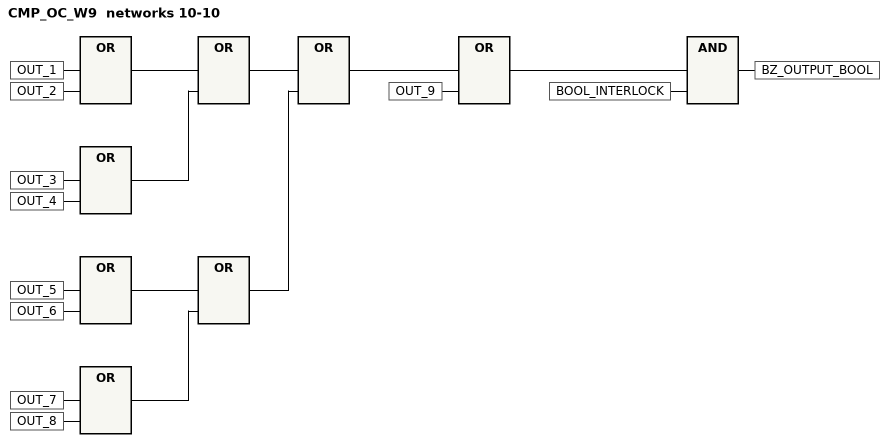
[picture p24: CMP_OC_W9 (FBD) networks 10-10]
_FBD_ (* Function Block Diagram *)
NETWORK 1
	OR(LT(WORD_1, 0), GT(WORD_1, 0)) => OUT_1
NETWORK 2
	OR(LT(WORD_2, 0), GT(WORD_2, 0)) => OUT_2
NETWORK 3
	OR(LT(WORD_3, 0), GT(WORD_3, 0)) => OUT_3
NETWORK 4
	OR(LT(WORD_4, 0), GT(WORD_4, 0)) => OUT_4
NETWORK 5
	OR(LT(WORD_5, 0), GT(WORD_5, 0)) => OUT_5
NETWORK 6
	OR(LT(WORD_6, 0), GT(WORD_6, 0)) => OUT_6
NETWORK 7
	OR(LT(WORD_7, 0), GT(WORD_7, 0)) => OUT_7
NETWORK 8
	OR(LT(WORD_8, 0), GT(WORD_8, 0)) => OUT_8
NETWORK 9
	OR(LT(WORD_9, 0), GT(WORD_9, 0)) => OUT_9
NETWORK 10
	AND(OR(OR(OR(OR(OUT_1, OUT_2), OR(OUT_3, OUT_4)), OR(OR(OUT_5, OUT_6), OR(OUT_7, OUT_8))), OUT_9), BOOL_INTERLOCK) => BZ_OUTPUT_BOOL
_END_FBD_
(* the same logic as Structured Text *)
(* Network 1 *)
OUT_1 := (WORD_1 < 0) OR (WORD_1 > 0);
(* Network 2 *)
OUT_2 := (WORD_2 < 0) OR (WORD_2 > 0);
(* Network 3 *)
OUT_3 := (WORD_3 < 0) OR (WORD_3 > 0);
(* Network 4 *)
OUT_4 := (WORD_4 < 0) OR (WORD_4 > 0);
(* Network 5 *)
OUT_5 := (WORD_5 < 0) OR (WORD_5 > 0);
(* Network 6 *)
OUT_6 := (WORD_6 < 0) OR (WORD_6 > 0);
(* Network 7 *)
OUT_7 := (WORD_7 < 0) OR (WORD_7 > 0);
(* Network 8 *)
OUT_8 := (WORD_8 < 0) OR (WORD_8 > 0);
(* Network 9 *)
OUT_9 := (WORD_9 < 0) OR (WORD_9 > 0);
(* Network 10 *)
BZ_OUTPUT_BOOL := ((((OUT_1 OR OUT_2) OR (OUT_3 OR OUT_4)) OR ((OUT_5 OR OUT_6) OR (OUT_7 OR OUT_8))) OR OUT_9) AND BOOL_INTERLOCK;
END_FUNCTION_BLOCK

(* POU DOWN_COUNT_TIMER, LD *)
FUNCTIONBLOCK DOWN_COUNT_TIMER
VAR_INPUT
	BOOL_SIGNAL_IN: BOOL;
	BOOL_TIMER_RST: BOOL;
	INT_AUTO_RST: INT;
	INT_SV_SEC: INT;
END_VAR
VAR_OUTPUT
	SIGNAL_BOOL: BOOL;
	PV_SEC_INT: INT;
END_VAR
VAR
	DF_1: R_TRIG;
	DF_2: R_TRIG;
	M1: BOOL;
	M2: BOOL;

	T100: TON;
	T101: TON;
	M100: BOOL;
	M101: BOOL;
	M200: BOOL;

	M110: BOOL;
	M300: BOOL;
END_VAR
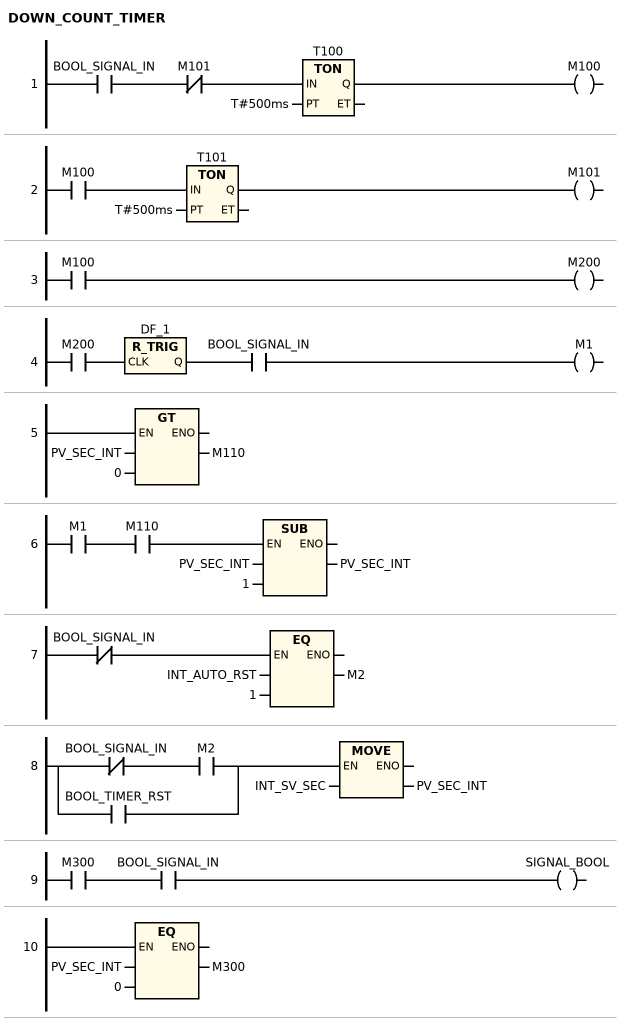
_LD_ (* Ladder Diagram *)
NETWORK 1
	[BOOL_SIGNAL_IN] - [/M101] - T100:TON(IN: *, PT: T#500ms) --- (M100)
NETWORK 2
	[M100] - T101:TON(IN: *, PT: T#500ms) --- (M101)
NETWORK 3
	[M100] --- (M200)
NETWORK 4
	[M200] - DF_1:R_TRIG(CLK: *) - [BOOL_SIGNAL_IN] --- (M1)
NETWORK 5
	*
		EN --- GT(PV_SEC_INT, 0) => M110
NETWORK 6
	[M1] - [M110]
		EN --- SUB(PV_SEC_INT, 1) => PV_SEC_INT
NETWORK 7
	[/BOOL_SIGNAL_IN]
		EN --- EQ(INT_AUTO_RST, 1) => M2
NETWORK 8
	{ [/BOOL_SIGNAL_IN] - [M2] | [BOOL_TIMER_RST] }
		EN --- MOVE(INT_SV_SEC) => PV_SEC_INT
NETWORK 9
	[M300] - [BOOL_SIGNAL_IN] --- (SIGNAL_BOOL)
NETWORK 10
	*
		EN --- EQ(PV_SEC_INT, 0) => M300
_END_LD_
(* the same logic as Structured Text *)
(* Network 1 *)
T100(IN := BOOL_SIGNAL_IN AND NOT M101, PT := T#500ms);
M100 := T100.Q;
(* Network 2 *)
T101(IN := M100, PT := T#500ms);
M101 := T101.Q;
(* Network 3 *)
M200 := M100;
(* Network 4 *)
DF_1(CLK := M200);
M1 := DF_1.Q AND BOOL_SIGNAL_IN;
(* Network 5 *)
M110 := PV_SEC_INT > 0;
(* Network 6 *)
IF M1 AND M110 THEN
	PV_SEC_INT := PV_SEC_INT - 1;
END_IF;
(* Network 7 *)
IF NOT BOOL_SIGNAL_IN THEN
	M2 := INT_AUTO_RST = 1;
END_IF;
(* Network 8 *)
IF NOT BOOL_SIGNAL_IN AND M2 OR BOOL_TIMER_RST THEN
	PV_SEC_INT := INT_SV_SEC;
END_IF;
(* Network 9 *)
SIGNAL_BOOL := M300 AND BOOL_SIGNAL_IN;
(* Network 10 *)
M300 := PV_SEC_INT = 0;
END_FUNCTION_BLOCK

(* POU CLOCK_PLS, LD *)
FUNCTION_BLOCK CLOCK_PLS
VAR_INPUT
	bCpStart			: BOOL;
	INT_TIME_ms 	: INT;

END_VAR
VAR_OUTPUT
	CLOCK_PLS_BOOL: BOOL;
END_VAR
VAR
	T0: TON;
	T1: TON;
	M0: BOOL;
	M1: BOOL;
	D0: TIME;
	D1: TIME;
END_VAR
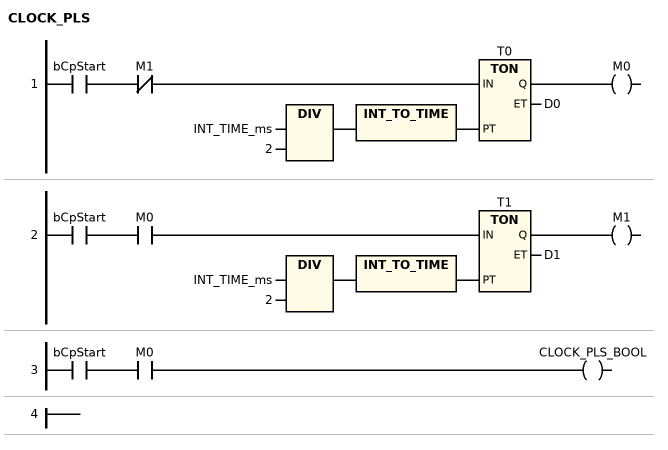
_LD_ (* Ladder Diagram *)
NETWORK 1
	[bCpStart] - [/M1] - T0:TON(IN: *, PT: INT_TO_TIME(DIV(INT_TIME_ms, 2)), ET => D0) --- (M0)
NETWORK 2
	[bCpStart] - [M0] - T1:TON(IN: *, PT: INT_TO_TIME(DIV(INT_TIME_ms, 2)), ET => D1) --- (M1)
NETWORK 3
	[bCpStart] - [M0] --- (CLOCK_PLS_BOOL)
NETWORK 4
	*
_END_LD_
(* the same logic as Structured Text *)
(* Network 1 *)
T0(IN := bCpStart AND NOT M1, PT := INT_TO_TIME(INT_TIME_ms / 2));
D0 := T0.ET;
M0 := T0.Q;
(* Network 2 *)
T1(IN := bCpStart AND M0, PT := INT_TO_TIME(INT_TIME_ms / 2));
D1 := T1.ET;
M1 := T1.Q;
(* Network 3 *)
CLOCK_PLS_BOOL := bCpStart AND M0;
(* Network 4 *)
END_FUNCTION_BLOCK

(* POU DC_PID_FB, LD *)
FUNCTION_BLOCK DC_PID_FB
VAR_INPUT
	BOOL_LOW_FLOW_EN : BOOL;
	INT_HIGH_FLOW_LPM : INT;
	INT_LOW_FLOW_LPM : INT;
	INT_H_L_FLOW_RATIO : INT;
	INT_D1_LPM : INT;
	INT_D2_LPM : INT;
	INT_D3_LPM : INT;
	INT_D4_RAW : INT;
	INT_D5_RAW : INT;
	INT_D6_RAW : INT;
	INT_D1_RATIO : INT;
	INT_D2_RATIO : INT;
	INT_D3_RATIO : INT;
	INT_D4_RATIO : INT;
	INT_D5_RATIO : INT;
	INT_D6_RATIO : INT;

END_VAR

VAR_OUTPUT

	PID_FLOW_RAW : INT;
	D1_RAW_INT : INT;
	D2_RAW_INT : INT;
	D3_RAW_INT : INT;
	D4_LPM_INT : INT;
	D5_LPM_INT : INT;
	D6_LPM_INT : INT;

END_VAR
VAR
	D5EN: BOOL;
	D4EN: BOOL;
	D6EN: BOOL;
	D4REN: BOOL;
	D5REN: BOOL;
	D6REN: BOOL;
END_VAR

(*

Thats 2 program in one function block

1st Program:- 
- Let user able to select High/low flow by trigger bit "BOOL_LOW_FLOW_EN"

	Sequence detail: 
	-If "BOOL_LOW_FLOW_EN" OFF, "INT_HIGH_FLOW_LPM" will MULTIPLY "INT_H_L_FLOW_RATIO" then Feed into "PID_FLOW_RAW".
	-If "BOOL_LOW_FLOW_EN" ON, "INT_LOW_FLOW_LPM" will MULTIPLY "INT_H_L_FLOW_RATIO" then Feed into "PID_FLOW_RAW".
	-"PID_FLOW_RAW should connect direct to ANALOG OUTPUT CARD CHANNEL.


2nd Program:-
-Become Converter. Able to convert 3 types of LPM reading to RAW reading by MULTIPLY the preset RATIO.
-Become Converter. Able to convert 3 types of RAW reading to LPM reading by DIVIDE the preset RATIO.

	Sequence detail:
	-Once detected INT_D1_LPM have value (Not "0") and INT_D1_RATIO have value (Not "0") -> Program will enable and MULTIPLY "INT_D1_LPM" with "INT_D1_RATIO" and feed to "D1_RAW_INT"
	-INT_D2_LPM, INT_D2_RATIO and D2_RAW_INT function same as above (D1)
	-INT_D3_LPM, INT_D3_RATIO and D3_RAW_INT function same as above (D1)
	-Once detected INT_D4_RAW have value (Not "0") and INT_D4_RATIO have value (Not "0") -> Program will enable and DIVIDE "INT_D4_RAW" with "INT_D4_RATIO" and feed to "D4_LPM_INT"
	-INT_D5_RAW, INT_D5_RATIO and D5_LPM_INT function same as above (D4)
	-INT_D6_RAW, INT_D6_RATIO and D6_LPM_INT function same as above (D4)

*)
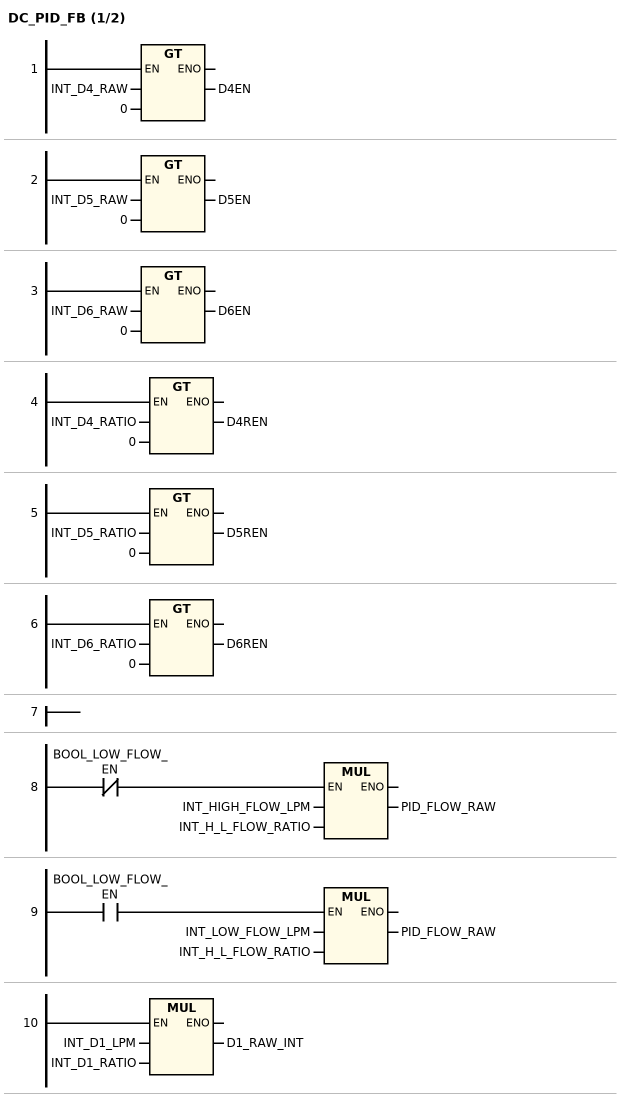
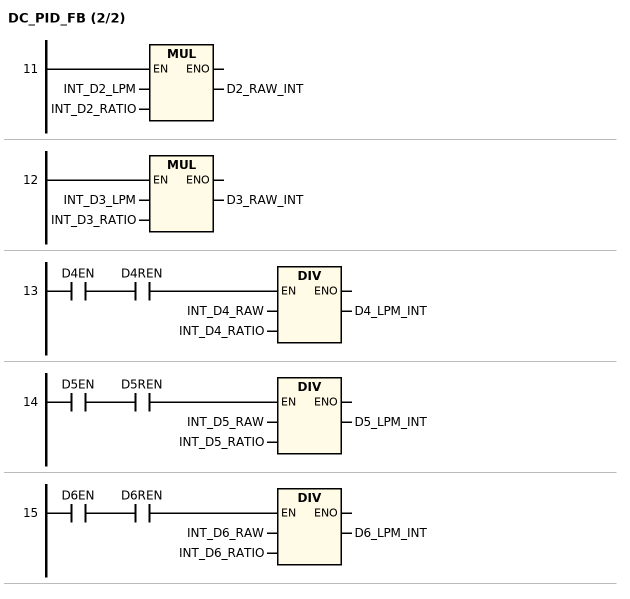
_LD_ (* Ladder Diagram *)
NETWORK 1
	*
		EN --- GT(INT_D4_RAW, 0) => D4EN
NETWORK 2
	*
		EN --- GT(INT_D5_RAW, 0) => D5EN
NETWORK 3
	*
		EN --- GT(INT_D6_RAW, 0) => D6EN
NETWORK 4
	*
		EN --- GT(INT_D4_RATIO, 0) => D4REN
NETWORK 5
	*
		EN --- GT(INT_D5_RATIO, 0) => D5REN
NETWORK 6
	*
		EN --- GT(INT_D6_RATIO, 0) => D6REN
NETWORK 7
	*
NETWORK 8
	[/BOOL_LOW_FLOW_EN]
		EN --- MUL(INT_HIGH_FLOW_LPM, INT_H_L_FLOW_RATIO) => PID_FLOW_RAW
NETWORK 9
	[BOOL_LOW_FLOW_EN]
		EN --- MUL(INT_LOW_FLOW_LPM, INT_H_L_FLOW_RATIO) => PID_FLOW_RAW
NETWORK 10
	*
		EN --- MUL(INT_D1_LPM, INT_D1_RATIO) => D1_RAW_INT
NETWORK 11
	*
		EN --- MUL(INT_D2_LPM, INT_D2_RATIO) => D2_RAW_INT
NETWORK 12
	*
		EN --- MUL(INT_D3_LPM, INT_D3_RATIO) => D3_RAW_INT
NETWORK 13
	[D4EN] - [D4REN]
		EN --- DIV(INT_D4_RAW, INT_D4_RATIO) => D4_LPM_INT
NETWORK 14
	[D5EN] - [D5REN]
		EN --- DIV(INT_D5_RAW, INT_D5_RATIO) => D5_LPM_INT
NETWORK 15
	[D6EN] - [D6REN]
		EN --- DIV(INT_D6_RAW, INT_D6_RATIO) => D6_LPM_INT
_END_LD_
(* the same logic as Structured Text *)
(* Network 1 *)
D4EN := INT_D4_RAW > 0;
(* Network 2 *)
D5EN := INT_D5_RAW > 0;
(* Network 3 *)
D6EN := INT_D6_RAW > 0;
(* Network 4 *)
D4REN := INT_D4_RATIO > 0;
(* Network 5 *)
D5REN := INT_D5_RATIO > 0;
(* Network 6 *)
D6REN := INT_D6_RATIO > 0;
(* Network 7 *)
(* Network 8 *)
IF NOT BOOL_LOW_FLOW_EN THEN
	PID_FLOW_RAW := INT_HIGH_FLOW_LPM * INT_H_L_FLOW_RATIO;
END_IF;
(* Network 9 *)
IF BOOL_LOW_FLOW_EN THEN
	PID_FLOW_RAW := INT_LOW_FLOW_LPM * INT_H_L_FLOW_RATIO;
END_IF;
(* Network 10 *)
D1_RAW_INT := INT_D1_LPM * INT_D1_RATIO;
(* Network 11 *)
D2_RAW_INT := INT_D2_LPM * INT_D2_RATIO;
(* Network 12 *)
D3_RAW_INT := INT_D3_LPM * INT_D3_RATIO;
(* Network 13 *)
IF D4EN AND D4REN THEN
	D4_LPM_INT := INT_D4_RAW / INT_D4_RATIO;
END_IF;
(* Network 14 *)
IF D5EN AND D5REN THEN
	D5_LPM_INT := INT_D5_RAW / INT_D5_RATIO;
END_IF;
(* Network 15 *)
IF D6EN AND D6REN THEN
	D6_LPM_INT := INT_D6_RAW / INT_D6_RATIO;
END_IF;
END_FUNCTION_BLOCK

(* POU EQ_GT, LD *)
FUNCTION_BLOCK EQ_GT
VAR_INPUT
	INT_SOURCE_A: INT;
	INT_SOURCE_B: INT;
END_VAR
VAR_OUTPUT
	SIGNAL_BOOL: BOOL;
END_VAR
VAR
	M0: BOOL;
	M1: BOOL;
END_VAR
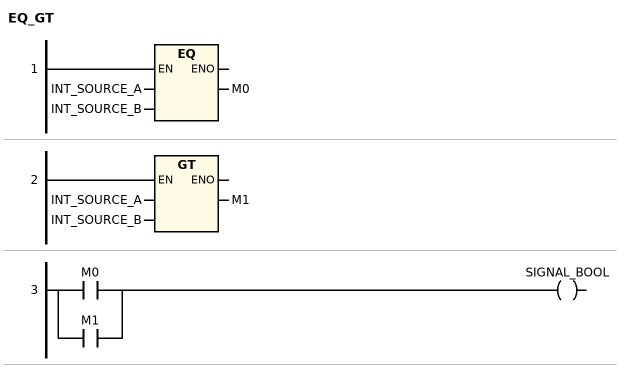
_LD_ (* Ladder Diagram *)
NETWORK 1
	*
		EN --- EQ(INT_SOURCE_A, INT_SOURCE_B) => M0
NETWORK 2
	*
		EN --- GT(INT_SOURCE_A, INT_SOURCE_B) => M1
NETWORK 3
	{ [M0] | [M1] } --- (SIGNAL_BOOL)
_END_LD_
(* the same logic as Structured Text *)
(* Network 1 *)
M0 := INT_SOURCE_A = INT_SOURCE_B;
(* Network 2 *)
M1 := INT_SOURCE_A > INT_SOURCE_B;
(* Network 3 *)
SIGNAL_BOOL := M0 OR M1;
END_FUNCTION_BLOCK

(* POU EQ_LT, LD *)
FUNCTION_BLOCK EQ_LT
VAR_INPUT
	INT_SOURCE_A:INT;
	INT_SOURCE_B:INT;
END_VAR
VAR_OUTPUT
	SIGNAL_BOOL:BOOL;
END_VAR
VAR
	M0: BOOL;
	M1: BOOL;
END_VAR
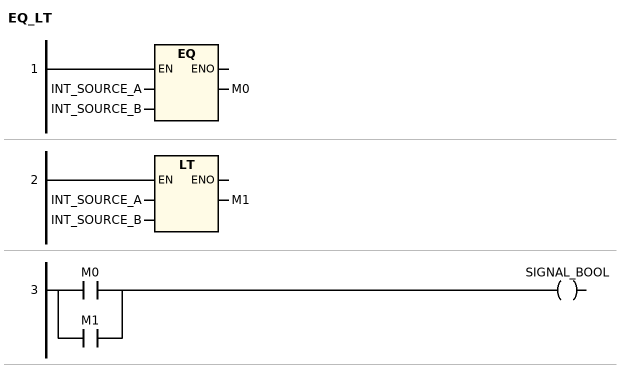
_LD_ (* Ladder Diagram *)
NETWORK 1
	*
		EN --- EQ(INT_SOURCE_A, INT_SOURCE_B) => M0
NETWORK 2
	*
		EN --- LT(INT_SOURCE_A, INT_SOURCE_B) => M1
NETWORK 3
	{ [M0] | [M1] } --- (SIGNAL_BOOL)
_END_LD_
(* the same logic as Structured Text *)
(* Network 1 *)
M0 := INT_SOURCE_A = INT_SOURCE_B;
(* Network 2 *)
M1 := INT_SOURCE_A < INT_SOURCE_B;
(* Network 3 *)
SIGNAL_BOOL := M0 OR M1;
END_FUNCTION_BLOCK

(* POU GUYSON_AI_CTRL, LD *)
FUNCTION_BLOCK GUYSON_AI_CTRL
VAR_INPUT

	BOOL_ST :BOOL; (*Analog Data Collection Start Bit*)
	INT_M1_AI :INT; (*Guyson Generator Master 1 Analog Input Data*)
	INT_M2_AI :INT; (*Guyson Generator Master 2 Analog Input Data*)
	TIME_REFRESH :TIME; (*Refresh Time assigned*)
	TIME_DATA_COLLECT :TIME; (*Delay time for data collection for stability improvement, This data must be ALWAYS "Half" or below from "TIME_REFRESH" SetPoint *)

END_VAR

VAR_OUTPUT

	M1CH1_INT :INT; (*ANALOG READING OF MASTER1-CHANNEL1*)
	M1CH2_INT :INT; (*ANALOG READING OF MASTER1-CHANNEL2*)
	S1CH1_INT :INT; (*ANALOG READING OF SLAVE1-CHANNEL1*)
	M2CH1_INT :INT; (*ANALOG READING OF MASTER2-CHANNEL1*)
	M2CH2_INT :INT; (*ANALOG READING OF MASTER2-CHANNEL2*)
	S2CH1_INT :INT; (*ANALOG READING OF SLAVE2-CHANNEL1*)
	M1_PIN1_DO_BOOL :BOOL; (*GUYSON MASTER 1 SCADA CONNECTOR PIN 1 (A0) CONNECTION OUTPUT FOR MODULE SELECTION*)
	M1_PIN7_DO_BOOL :BOOL; (*GUYSON MASTER 1 SCADA CONNECTOR PIN 7 (A3) CONNECTION OUTPUT FOR IDENTITY SELECTION*)
	M2_PIN1_DO_BOOL :BOOL; (*GUYSON MASTER 2 SCADA CONNECTOR PIN 1 (A0) CONNECTION OUTPUT FOR MODULE SELECTION*)
	M2_PIN7_DO_BOOL :BOOL; (*GUYSON MASTER 2 SCADA CONNECTOR PIN 7 (A3) CONNECTION OUTPUT FOR IDENTITY SELECTION*)
	IT1AOUT_BOOL: BOOL;
	IT2AOUT_BOOL: BOOL;
	IT3AOUT_BOOL: BOOL;
	IT1BOUT_BOOL: BOOL;
	IT2BOUT_BOOL: BOOL;
	IT3BOUT_BOOL: BOOL;





END_VAR
VAR
	IT1A: TON;
	IT2A: TON;
	IT3A: TON;
	IT1B: TON;
	IT2B: TON;
	IT3B: TON;


	M1CH1BOOLOUT: BOOL;
	M1CH2BOOLOUT: BOOL;
	S1CH1BOOLOUT: BOOL;
	M2CH1BOOLOUT: BOOL;
	M2CH2BOOLOUT: BOOL;
	S2CH1BOOLOUT: BOOL;

END_VAR
VAR (* helpers for the ST form of the networks *)
	_p1 : BOOL;
	_p2 : BOOL;
	_p3 : BOOL;
END_VAR
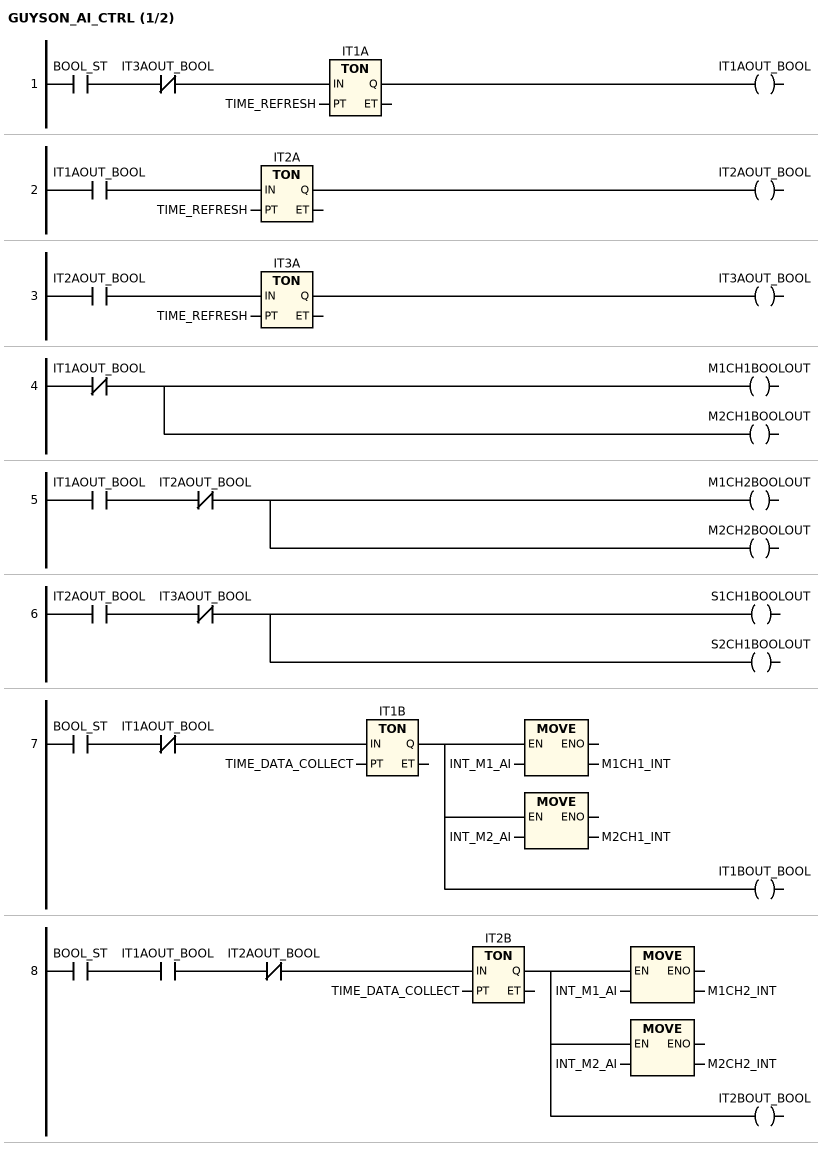
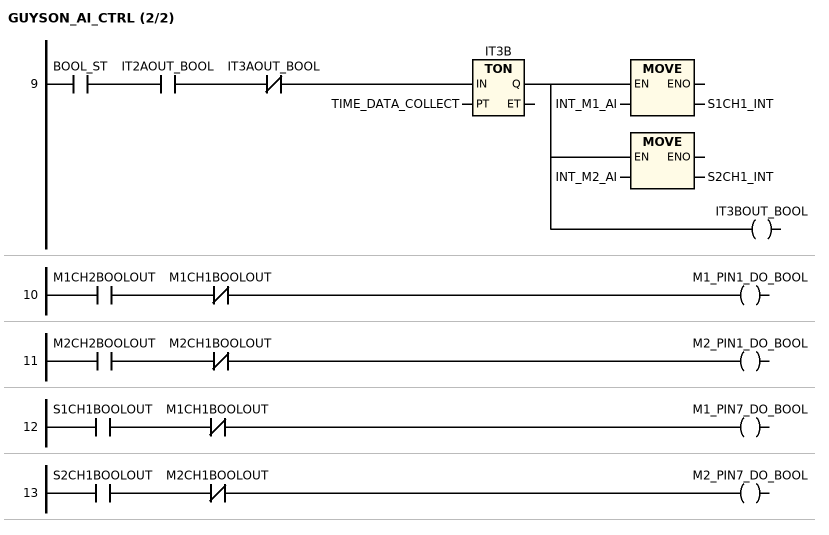
_LD_ (* Ladder Diagram *)
NETWORK 1
	[BOOL_ST] - [/IT3AOUT_BOOL] - IT1A:TON(IN: *, PT: TIME_REFRESH) --- (IT1AOUT_BOOL)
NETWORK 2
	[IT1AOUT_BOOL] - IT2A:TON(IN: *, PT: TIME_REFRESH) --- (IT2AOUT_BOOL)
NETWORK 3
	[IT2AOUT_BOOL] - IT3A:TON(IN: *, PT: TIME_REFRESH) --- (IT3AOUT_BOOL)
NETWORK 4
	[/IT1AOUT_BOOL] --- (M1CH1BOOLOUT) (M2CH1BOOLOUT)
NETWORK 5
	[IT1AOUT_BOOL] - [/IT2AOUT_BOOL] --- (M1CH2BOOLOUT) (M2CH2BOOLOUT)
NETWORK 6
	[IT2AOUT_BOOL] - [/IT3AOUT_BOOL] --- (S1CH1BOOLOUT) (S2CH1BOOLOUT)
NETWORK 7
	[BOOL_ST] - [/IT1AOUT_BOOL] - IT1B:TON(IN: *, PT: TIME_DATA_COLLECT) --- (IT1BOUT_BOOL)
		EN --- MOVE(INT_M1_AI) => M1CH1_INT
		EN --- MOVE(INT_M2_AI) => M2CH1_INT
NETWORK 8
	[BOOL_ST] - [IT1AOUT_BOOL] - [/IT2AOUT_BOOL] - IT2B:TON(IN: *, PT: TIME_DATA_COLLECT) --- (IT2BOUT_BOOL)
		EN --- MOVE(INT_M1_AI) => M1CH2_INT
		EN --- MOVE(INT_M2_AI) => M2CH2_INT
NETWORK 9
	[BOOL_ST] - [IT2AOUT_BOOL] - [/IT3AOUT_BOOL] - IT3B:TON(IN: *, PT: TIME_DATA_COLLECT) --- (IT3BOUT_BOOL)
		EN --- MOVE(INT_M1_AI) => S1CH1_INT
		EN --- MOVE(INT_M2_AI) => S2CH1_INT
NETWORK 10
	[M1CH2BOOLOUT] - [/M1CH1BOOLOUT] --- (M1_PIN1_DO_BOOL)
NETWORK 11
	[M2CH2BOOLOUT] - [/M2CH1BOOLOUT] --- (M2_PIN1_DO_BOOL)
NETWORK 12
	[S1CH1BOOLOUT] - [/M1CH1BOOLOUT] --- (M1_PIN7_DO_BOOL)
NETWORK 13
	[S2CH1BOOLOUT] - [/M2CH1BOOLOUT] --- (M2_PIN7_DO_BOOL)
_END_LD_
(* the same logic as Structured Text *)
(* Network 1 *)
IT1A(IN := BOOL_ST AND NOT IT3AOUT_BOOL, PT := TIME_REFRESH);
IT1AOUT_BOOL := IT1A.Q;
(* Network 2 *)
IT2A(IN := IT1AOUT_BOOL, PT := TIME_REFRESH);
IT2AOUT_BOOL := IT2A.Q;
(* Network 3 *)
IT3A(IN := IT2AOUT_BOOL, PT := TIME_REFRESH);
IT3AOUT_BOOL := IT3A.Q;
(* Network 4 *)
M1CH1BOOLOUT := NOT IT1AOUT_BOOL;
M2CH1BOOLOUT := M1CH1BOOLOUT;
(* Network 5 *)
M1CH2BOOLOUT := IT1AOUT_BOOL AND NOT IT2AOUT_BOOL;
M2CH2BOOLOUT := M1CH2BOOLOUT;
(* Network 6 *)
S1CH1BOOLOUT := IT2AOUT_BOOL AND NOT IT3AOUT_BOOL;
S2CH1BOOLOUT := S1CH1BOOLOUT;
(* Network 7 *)
IT1B(IN := BOOL_ST AND NOT IT1AOUT_BOOL, PT := TIME_DATA_COLLECT);
_p1 := IT1B.Q;
IF _p1 THEN
	M1CH1_INT := INT_M1_AI;
	M2CH1_INT := INT_M2_AI;
END_IF;
IT1BOUT_BOOL := _p1;
(* Network 8 *)
IT2B(IN := BOOL_ST AND IT1AOUT_BOOL AND NOT IT2AOUT_BOOL, PT := TIME_DATA_COLLECT);
_p2 := IT2B.Q;
IF _p2 THEN
	M1CH2_INT := INT_M1_AI;
	M2CH2_INT := INT_M2_AI;
END_IF;
IT2BOUT_BOOL := _p2;
(* Network 9 *)
IT3B(IN := BOOL_ST AND IT2AOUT_BOOL AND NOT IT3AOUT_BOOL, PT := TIME_DATA_COLLECT);
_p3 := IT3B.Q;
IF _p3 THEN
	S1CH1_INT := INT_M1_AI;
	S2CH1_INT := INT_M2_AI;
END_IF;
IT3BOUT_BOOL := _p3;
(* Network 10 *)
M1_PIN1_DO_BOOL := M1CH2BOOLOUT AND NOT M1CH1BOOLOUT;
(* Network 11 *)
M2_PIN1_DO_BOOL := M2CH2BOOLOUT AND NOT M2CH1BOOLOUT;
(* Network 12 *)
M1_PIN7_DO_BOOL := S1CH1BOOLOUT AND NOT M1CH1BOOLOUT;
(* Network 13 *)
M2_PIN7_DO_BOOL := S2CH1BOOLOUT AND NOT M2CH1BOOLOUT;
END_FUNCTION_BLOCK

(* POU GUYSON_AI_RawToWatt, ST *)
FUNCTION_BLOCK GUYSON_AI_RawToWatt
VAR_INPUT

	iAI1raw : INT;				(* 1st Raw Data From Analog Input*)
	iAI2raw : INT;				(* 2nd Raw Data From Analog Input*)
	iAI3raw : INT;				(* 3rd Raw Data From Analog Input*)
	iAI4raw : INT;				(* 4th Raw Data From Analog Input*)
	iAI5raw : INT;				(* 5th Raw Data From Analog Input*)
	iAI6raw : INT;				(* 6th Raw Data From Analog Input*)
	PercentBase : BOOL;		(* The PV will shown Percentage if this Bit is "ON"*)
	WattBase : BOOL;			(* The PV will shown Wattage if this Bit is "ON"*)
	MaxWatt : INT;			(* Defined Max Watt of Generator, Usually is 700W*)

END_VAR
VAR_OUTPUT

	iAI1Value : INT;			(*PV for 1st Data, either Watt or Percent is depend on Base Setting*)
	iAI2Value : INT;			(*PV for 2nd Data, either Watt or Percent is depend on Base Setting*)
	iAI3Value : INT;			(*PV for 3rd Data, either Watt or Percent is depend on Base Setting*)
	iAI4Value : INT;			(*PV for 4th Data, either Watt or Percent is depend on Base Setting*)
	iAI5Value : INT;			(*PV for 5th Data, either Watt or Percent is depend on Base Setting*)
	iAI6Value : INT;			(*PV for 6th Data, either Watt or Percent is depend on Base Setting*)

END_VAR
VAR
	iAI1f: LREAL;
	iAI2f: LREAL;
	iAI3f: LREAL;
	iAI4f: LREAL;
	iAI5f: LREAL;
	iAI6f: LREAL;

	iAI1_Wf: LREAL;
	iAI2_Wf: LREAL;
	iAI3_Wf: LREAL;
	iAI4_Wf: LREAL;
	iAI5_Wf: LREAL;
	iAI6_Wf: LREAL;

	n : INT;

	WRatio: INT;
END_VAR
iAI1f := INT_TO_LREAL (iAI1raw);
iAI2f := INT_TO_LREAL (iAI2raw);
iAI3f := INT_TO_LREAL (iAI3raw);
iAI4f := INT_TO_LREAL (iAI4raw);
iAI5f := INT_TO_LREAL (iAI5raw);
iAI6f := INT_TO_LREAL (iAI6raw);


(*Program to select Watt Base or Percent Base*)

IF PercentBase AND NOT WattBase THEN
n := 11;
END_IF

IF WattBase AND NOT PercentBase THEN
n := 10;
END_IF

IF NOT PercentBase AND NOT WattBase THEN
n := 0;
END_IF

IF PercentBase AND WattBase THEN
n:= 0;
END_IF

CASE n OF

0:; (*No Calculation*)


10: (*Watt Base Calculation *)

iAI1_Wf	:= (iAI1f / 3276.7) * (iAI1f / 3276.7) *20;
iAI2_Wf	:= (iAI2f / 3276.7) * (iAI2f / 3276.7) *20;
iAI3_Wf	:= (iAI3f / 3276.7) * (iAI3f / 3276.7) *20;
iAI4_Wf	:= (iAI4f / 3276.7) * (iAI4f / 3276.7) *20;
iAI5_Wf	:= (iAI5f / 3276.7) * (iAI5f / 3276.7) *20;
iAI6_Wf	:= (iAI6f / 3276.7) * (iAI6f / 3276.7) *20;


11: (*Percent Base Calculation*)


WRatio := MaxWatt/100;


iAI1_Wf	:= ((iAI1f / 3276.7) * (iAI1f / 3276.7) *20)/WRatio;
iAI2_Wf	:= ((iAI2f / 3276.7) * (iAI2f / 3276.7) *20)/WRatio;
iAI3_Wf	:= ((iAI3f / 3276.7) * (iAI3f / 3276.7) *20)/WRatio;
iAI4_Wf	:= ((iAI4f / 3276.7) * (iAI4f / 3276.7) *20)/WRatio;
iAI5_Wf	:= ((iAI5f / 3276.7) * (iAI5f / 3276.7) *20)/WRatio;
iAI6_Wf	:= ((iAI6f / 3276.7) * (iAI6f / 3276.7) *20)/WRatio;

END_CASE

iAI1Value := LREAL_TO_INT (iAI1_Wf);
iAI2Value := LREAL_TO_INT (iAI2_Wf);
iAI3Value := LREAL_TO_INT (iAI3_Wf);
iAI4Value := LREAL_TO_INT (iAI4_Wf);
iAI5Value := LREAL_TO_INT (iAI5_Wf);
iAI6Value := LREAL_TO_INT (iAI6_Wf);
END_FUNCTION_BLOCK

(* POU GUYSON_AI_WattToRaw, ST *)
FUNCTION_BLOCK GUYSON_AI_WattToRaw
VAR_INPUT

	iAI1SP : INT;			(* 1st SetPoint Data*)
	iAI2SP : INT;			(* 2nd SetPoint Data*)
	iAI3SP : INT;			(* 3rd SetPoint Data*)
	iAI4SP : INT;			(* 4th SetPoint Data*)
	iAI5SP : INT;			(* 5th SetPoint Data*)
	iAI6SP : INT;			(* 6th SetPoint Data*)
	PercentBase : BOOL;	(* The PV will shown Percentage if this Bit is "ON"*)
	WattBase: BOOL;		(* The PV will shown Wattage if this Bit is "ON"*)
	MinSP : INT;			(* Define Min SetPoint Input, if SP set below this value, the PV will become "0"*)
	MaxSP : INT;			(* Define Max SetPoint Input, if SP set Greater than value, the PV will become "0"*)
	MaxWatt : INT;		(* Defined Max Watt of Generator, Usually is 700W*)


END_VAR

VAR_OUTPUT

	iAI1raw : INT;			(*1st Raw Data to feed to Analog Output Card for Ultrasonic Generator Power Control*)
	iAI2raw : INT;			(*2nd Raw Data to feed to Analog Output Card for Ultrasonic Generator Power Control*)
	iAI3raw : INT;			(*3rd Raw Data to feed to Analog Output Card for Ultrasonic Generator Power Control*)
	iAI4raw : INT;			(*4th Raw Data to feed to Analog Output Card for Ultrasonic Generator Power Control*)
	iAI5raw : INT;			(*5th Raw Data to feed to Analog Output Card for Ultrasonic Generator Power Control*)
	iAI6raw : INT;			(*6th Raw Data to feed to Analog Output Card for Ultrasonic Generator Power Control*)

END_VAR
VAR
	iAI1f: LREAL;
	iAI2f: LREAL;
	iAI3f: LREAL;
	iAI4f: LREAL;
	iAI5f: LREAL;
	iAI6f: LREAL;

	iAI1_Wf: LREAL;
	iAI2_Wf: LREAL;
	iAI3_Wf: LREAL;
	iAI4_Wf: LREAL;
	iAI5_Wf: LREAL;
	iAI6_Wf: LREAL;

	n : INT;
	WRatio: INT;
END_VAR
(*Set Min and Max Limit for Watt input*)
(*Convert INT to LREAL for Calculation*)

IF iAI1SP>=MinSP AND iAI1SP<=MaxSP THEN
iAI1_Wf := INT_TO_LREAL (iAI1SP);
ELSE iAI1_Wf := 0;
END_IF

IF iAI2SP>=MinSP AND iAI2SP<=MaxSP THEN
iAI2_Wf := INT_TO_LREAL (iAI2SP);
ELSE iAI2_Wf := 0;
END_IF

IF iAI3SP>=MinSP AND iAI3SP<=MaxSP THEN
iAI3_Wf := INT_TO_LREAL (iAI3SP);
ELSE iAI3_Wf := 0;
END_IF

IF iAI4SP>=MinSP AND iAI4SP<=MaxSP THEN
iAI4_Wf := INT_TO_LREAL (iAI4SP);
ELSE iAI4_Wf := 0;
END_IF

IF iAI5SP>=MinSP AND iAI5SP<=MaxSP THEN
iAI5_Wf := INT_TO_LREAL (iAI5SP);
ELSE iAI5_Wf := 0;
END_IF

IF iAI6SP>=MinSP AND iAI6SP<=MaxSP THEN
iAI6_Wf := INT_TO_LREAL (iAI6SP);
ELSE iAI6_Wf := 0;
END_IF

(*Program to select Watt Base or Percent Base*)

IF PercentBase AND NOT WattBase THEN
n := 11;
END_IF

IF WattBase AND NOT PercentBase THEN
n := 10;
END_IF

IF NOT PercentBase AND NOT WattBase THEN
n := 0;
END_IF

IF PercentBase AND WattBase THEN
n:= 0;
END_IF



CASE n OF

0:;	(*No Calculation Apply*)

10:	(*Watt Base Calculation*)

WRatio := MaxWatt/100;


	iAI1f	:= iAI1_Wf/WRatio*327.67;
	iAI2f	:= iAI2_Wf/WRatio*327.67;
	iAI3f	:= iAI3_Wf/WRatio*327.67;
	iAI4f	:= iAI4_Wf/WRatio*327.67;
	iAI5f	:= iAI5_Wf/WRatio*327.67;
	iAI6f	:= iAI6_Wf/WRatio*327.67;


(*	iAI1f	:= (SQRT(iAI1_Wf/20))*3276.7;
	iAI2f	:= (SQRT(iAI2_Wf/20))*3276.7;
	iAI3f	:= (SQRT(iAI3_Wf/20))*3276.7;
	iAI4f	:= (SQRT(iAI4_Wf/20))*3276.7;
	iAI5f	:= (SQRT(iAI5_Wf/20))*3276.7;
	iAI6f	:= (SQRT(iAI6_Wf/20))*3276.7;
*)

11: 	(*% Base Calculation*)

	iAI1f	:= iAI1_Wf*327.67;
	iAI2f	:= iAI2_Wf*327.67;
	iAI3f	:= iAI3_Wf*327.67;
	iAI4f	:= iAI4_Wf*327.67;
	iAI5f	:= iAI5_Wf*327.67;
	iAI6f	:= iAI6_Wf*327.67;

END_CASE

iAI1raw := LREAL_TO_INT (iAI1f);
iAI2raw := LREAL_TO_INT (iAI2f);
iAI3raw := LREAL_TO_INT (iAI3f);
iAI4raw := LREAL_TO_INT (iAI4f);
iAI5raw := LREAL_TO_INT (iAI5f);
iAI6raw := LREAL_TO_INT (iAI6f);
END_FUNCTION_BLOCK

(* POU GUYSON_PRG_SEL, FBD *)
FUNCTION_BLOCK GUYSON_PRG_SEL
VAR_INPUT

	US_ON_BOOL		:BOOL; 		(*ULTRASONIC ON/OFF BIT*)
	PRG_ADD_INT		:INT;		(*PROGRAM ADDRESS*)


END_VAR
VAR_OUTPUT

	BOOL_US_BIT1		:BOOL; 		(*ULTRASONIC EXT1*)
	BOOL_US_BIT2		:BOOL; 		(*ULTRASONIC EXT2*)
	BOOL_US_BIT3		:BOOL; 		(*ULTRASONIC EXT3*)


END_VAR
VAR
END_VAR
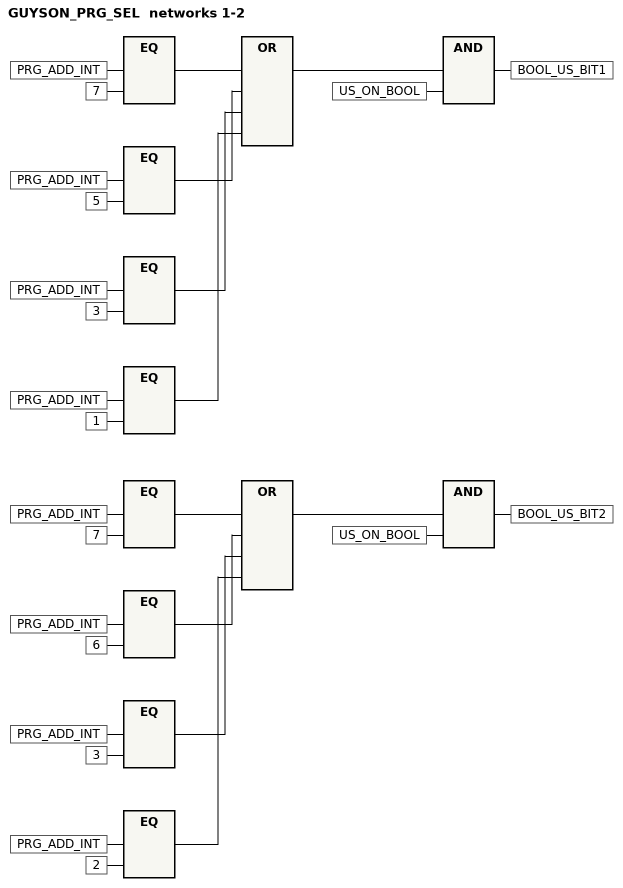
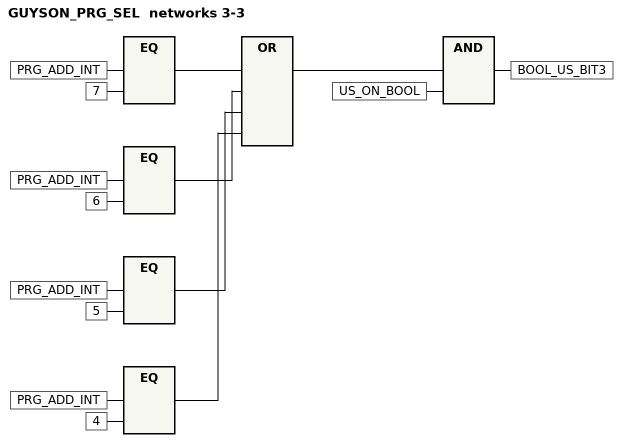
_FBD_ (* Function Block Diagram *)
NETWORK 1
	AND(OR(EQ(PRG_ADD_INT, 7), EQ(PRG_ADD_INT, 5), EQ(PRG_ADD_INT, 3), EQ(PRG_ADD_INT, 1)), US_ON_BOOL) => BOOL_US_BIT1
NETWORK 2
	AND(OR(EQ(PRG_ADD_INT, 7), EQ(PRG_ADD_INT, 6), EQ(PRG_ADD_INT, 3), EQ(PRG_ADD_INT, 2)), US_ON_BOOL) => BOOL_US_BIT2
NETWORK 3
	AND(OR(EQ(PRG_ADD_INT, 7), EQ(PRG_ADD_INT, 6), EQ(PRG_ADD_INT, 5), EQ(PRG_ADD_INT, 4)), US_ON_BOOL) => BOOL_US_BIT3
_END_FBD_
(* the same logic as Structured Text *)
(* Network 1 *)
BOOL_US_BIT1 := ((PRG_ADD_INT = 7) OR (PRG_ADD_INT = 5) OR (PRG_ADD_INT = 3) OR (PRG_ADD_INT = 1)) AND US_ON_BOOL;
(* Network 2 *)
BOOL_US_BIT2 := ((PRG_ADD_INT = 7) OR (PRG_ADD_INT = 6) OR (PRG_ADD_INT = 3) OR (PRG_ADD_INT = 2)) AND US_ON_BOOL;
(* Network 3 *)
BOOL_US_BIT3 := ((PRG_ADD_INT = 7) OR (PRG_ADD_INT = 6) OR (PRG_ADD_INT = 5) OR (PRG_ADD_INT = 4)) AND US_ON_BOOL;
END_FUNCTION_BLOCK

(* POU INDIRECT_FN, LD *)
FUNCTION_BLOCK INDIRECT_FN
VAR_INPUT
	BOOL_SV_PB: BOOL;		(*SAVE PB (TS)*)
	BOOL_LD_PB: BOOL;			(*LOAD PB (TS)*)
	INT_P_NO: INT;		(*PROGRAM NO (TS) 1~10*)
	INT_D00:INT;
	INT_D01:INT;
	INT_D02:INT;
	INT_D03:INT;
	INT_D04:INT;
	INT_D05:INT;
	INT_D06:INT;
	INT_D07:INT;
	INT_D08:INT;
	INT_D09:INT;
	INT_D10:INT;
	INT_D11:INT;
	INT_D12:INT;
	INT_D13:INT;
	INT_D14:INT;
	INT_D15:INT;
	INT_D16:INT;
	INT_D17:INT;
	INT_D18:INT;
	INT_D19:INT;
	INT_D20:INT;
	INT_D21:INT;
	INT_D22:INT;
	INT_D23:INT;
	INT_D24:INT;
	INT_D25:INT;
	INT_D26:INT;
	INT_D27:INT;
	INT_D28:INT;
	INT_D29:INT;
	INT_D30:INT;
	STG_STG1:STRING;
END_VAR
VAR_OUTPUT
	SV_PB_IND_BOOL:BOOL;
	LD_PB_IND_BOOL:BOOL;
	D00_INT:INT;
	D01_INT:INT;
	D02_INT:INT;
	D03_INT:INT;
	D04_INT:INT;
	D05_INT:INT;
	D06_INT:INT;
	D07_INT:INT;
	D08_INT:INT;
	D09_INT:INT;
	D10_INT:INT;
	D11_INT:INT;
	D12_INT:INT;
	D13_INT:INT;
	D14_INT:INT;
	D15_INT:INT;
	D16_INT:INT;
	D17_INT:INT;
	D18_INT:INT;
	D19_INT:INT;
	D20_INT:INT;
	D21_INT:INT;
	D22_INT:INT;
	D23_INT:INT;
	D24_INT:INT;
	D25_INT:INT;
	D26_INT:INT;
	D27_INT:INT;
	D28_INT:INT;
	D29_INT:INT;
	D30_INT:INT;
	STG1_STG:STRING;
END_VAR
VAR

	P1B: BOOL;
	P2B: BOOL;
	P3B: BOOL;
	P4B: BOOL;
	P5B: BOOL;
	P6B: BOOL;
	P7B: BOOL;
	P8B: BOOL;
	P9B: BOOL;
	P10B: BOOL;
	SV_HR: BOOL;
	SV_T: TON;
	SV_CR: BOOL;
	LD_HR: BOOL;
	LD_CR: BOOL;
	LD_T: TON;
	SV_DF: R_TRIG;
	SV_PLS: BOOL;
	LD_DF: R_TRIG;
	LD_PLS: BOOL;
	ALWAYS_ON: BOOL;
	TPC: TON;
	N0: BOOL;
	TPC1: TON;
	N1: BOOL;
	CNG_P_NO: INT;
	NPC: BOOL;		(*NON PROGRAM CHANGE*)
	PCDF: R_TRIG;
	PCTDF: BOOL;
	PCDFN: F_TRIG;
	PC_PLS: BOOL;
	SVPLS: R_TRIG;
	SV_PB_PLS: BOOL;
	LDPLS: R_TRIG;
	LD_PB_PLS: BOOL;
END_VAR
VAR PERSISTENT
	P01D00:INT;
	P01D01:INT;
	P01D02:INT;
	P01D03:INT;
	P01D04:INT;
	P01D05:INT;
	P01D06:INT;
	P01D07:INT;
	P01D08:INT;
	P01D09:INT;
	P01D10:INT;
	P01D11:INT;
	P01D12:INT;
	P01D13:INT;
	P01D14:INT;
	P01D15:INT;
	P01D16:INT;
	P01D17:INT;
	P01D18:INT;
	P01D19:INT;
	P01D20:INT;
	P01D21:INT;
	P01D22:INT;
	P01D23:INT;
	P01D24:INT;
	P01D25:INT;
	P01D26:INT;
	P01D27:INT;
	P01D28:INT;
	P01D29:INT;
	P01D30:INT;
	P01STG:STRING;
	P02D00:INT;
	P02D01:INT;
	P02D02:INT;
	P02D03:INT;
	P02D04:INT;
	P02D05:INT;
	P02D06:INT;
	P02D07:INT;
	P02D08:INT;
	P02D09:INT;
	P02D10:INT;
	P02D11:INT;
	P02D12:INT;
	P02D13:INT;
	P02D14:INT;
	P02D15:INT;
	P02D16:INT;
	P02D17:INT;
	P02D18:INT;
	P02D19:INT;
	P02D20:INT;
	P02D21:INT;
	P02D22:INT;
	P02D23:INT;
	P02D24:INT;
	P02D25:INT;
	P02D26:INT;
	P02D27:INT;
	P02D28:INT;
	P02D29:INT;
	P02D30:INT;
	P02STG:STRING;
	P03D00:INT;
	P03D01:INT;
	P03D02:INT;
	P03D03:INT;
	P03D04:INT;
	P03D05:INT;
	P03D06:INT;
	P03D07:INT;
	P03D08:INT;
	P03D09:INT;
	P03D10:INT;
	P03D11:INT;
	P03D12:INT;
	P03D13:INT;
	P03D14:INT;
	P03D15:INT;
	P03D16:INT;
	P03D17:INT;
	P03D18:INT;
	P03D19:INT;
	P03D20:INT;
	P03D21:INT;
	P03D22:INT;
	P03D23:INT;
	P03D24:INT;
	P03D25:INT;
	P03D26:INT;
	P03D27:INT;
	P03D28:INT;
	P03D29:INT;
	P03D30:INT;
	P03STG:STRING;
	P04D00:INT;
	P04D01:INT;
	P04D02:INT;
	P04D03:INT;
	P04D04:INT;
	P04D05:INT;
	P04D06:INT;
	P04D07:INT;
	P04D08:INT;
	P04D09:INT;
	P04D10:INT;
	P04D11:INT;
	P04D12:INT;
	P04D13:INT;
	P04D14:INT;
	P04D15:INT;
	P04D16:INT;
	P04D17:INT;
	P04D18:INT;
	P04D19:INT;
	P04D20:INT;
	P04D21:INT;
	P04D22:INT;
	P04D23:INT;
	P04D24:INT;
	P04D25:INT;
	P04D26:INT;
	P04D27:INT;
	P04D28:INT;
	P04D29:INT;
	P04D30:INT;
	P04STG:STRING;
	P05D00:INT;
	P05D01:INT;
	P05D02:INT;
	P05D03:INT;
	P05D04:INT;
	P05D05:INT;
	P05D06:INT;
	P05D07:INT;
	P05D08:INT;
	P05D09:INT;
	P05D10:INT;
	P05D11:INT;
	P05D12:INT;
	P05D13:INT;
	P05D14:INT;
	P05D15:INT;
	P05D16:INT;
	P05D17:INT;
	P05D18:INT;
	P05D19:INT;
	P05D20:INT;
	P05D21:INT;
	P05D22:INT;
	P05D23:INT;
	P05D24:INT;
	P05D25:INT;
	P05D26:INT;
	P05D27:INT;
	P05D28:INT;
	P05D29:INT;
	P05D30:INT;
	P05STG:STRING;
	P06D00:INT;
	P06D01:INT;
	P06D02:INT;
	P06D03:INT;
	P06D04:INT;
	P06D05:INT;
	P06D06:INT;
	P06D07:INT;
	P06D08:INT;
	P06D09:INT;
	P06D10:INT;
	P06D11:INT;
	P06D12:INT;
	P06D13:INT;
	P06D14:INT;
	P06D15:INT;
	P06D16:INT;
	P06D17:INT;
	P06D18:INT;
	P06D19:INT;
	P06D20:INT;
	P06D21:INT;
	P06D22:INT;
	P06D23:INT;
	P06D24:INT;
	P06D25:INT;
	P06D26:INT;
	P06D27:INT;
	P06D28:INT;
	P06D29:INT;
	P06D30:INT;
	P06STG:STRING;
	P07D00:INT;
	P07D01:INT;
	P07D02:INT;
	P07D03:INT;
	P07D04:INT;
	P07D05:INT;
	P07D06:INT;
	P07D07:INT;
	P07D08:INT;
	P07D09:INT;
	P07D10:INT;
	P07D11:INT;
	P07D12:INT;
	P07D13:INT;
	P07D14:INT;
	P07D15:INT;
	P07D16:INT;
	P07D17:INT;
	P07D18:INT;
	P07D19:INT;
	P07D20:INT;
	P07D21:INT;
	P07D22:INT;
	P07D23:INT;
	P07D24:INT;
	P07D25:INT;
	P07D26:INT;
	P07D27:INT;
	P07D28:INT;
	P07D29:INT;
	P07D30:INT;
	P07STG:STRING;
	P08D00:INT;
	P08D01:INT;
	P08D02:INT;
	P08D03:INT;
	P08D04:INT;
	P08D05:INT;
	P08D06:INT;
	P08D07:INT;
	P08D08:INT;
	P08D09:INT;
	P08D10:INT;
	P08D11:INT;
	P08D12:INT;
	P08D13:INT;
	P08D14:INT;
	P08D15:INT;
	P08D16:INT;
	P08D17:INT;
	P08D18:INT;
	P08D19:INT;
	P08D20:INT;
	P08D21:INT;
	P08D22:INT;
	P08D23:INT;
	P08D24:INT;
	P08D25:INT;
	P08D26:INT;
	P08D27:INT;
	P08D28:INT;
	P08D29:INT;
	P08D30:INT;
	P08STG:STRING;
	P09D00:INT;
	P09D01:INT;
	P09D02:INT;
	P09D03:INT;
	P09D04:INT;
	P09D05:INT;
	P09D06:INT;
	P09D07:INT;
	P09D08:INT;
	P09D09:INT;
	P09D10:INT;
	P09D11:INT;
	P09D12:INT;
	P09D13:INT;
	P09D14:INT;
	P09D15:INT;
	P09D16:INT;
	P09D17:INT;
	P09D18:INT;
	P09D19:INT;
	P09D20:INT;
	P09D21:INT;
	P09D22:INT;
	P09D23:INT;
	P09D24:INT;
	P09D25:INT;
	P09D26:INT;
	P09D27:INT;
	P09D28:INT;
	P09D29:INT;
	P09D30:INT;
	P09STG:STRING;
	P10D00:INT;
	P10D01:INT;
	P10D02:INT;
	P10D03:INT;
	P10D04:INT;
	P10D05:INT;
	P10D06:INT;
	P10D07:INT;
	P10D08:INT;
	P10D09:INT;
	P10D10:INT;
	P10D11:INT;
	P10D12:INT;
	P10D13:INT;
	P10D14:INT;
	P10D15:INT;
	P10D16:INT;
	P10D17:INT;
	P10D18:INT;
	P10D19:INT;
	P10D20:INT;
	P10D21:INT;
	P10D22:INT;
	P10D23:INT;
	P10D24:INT;
	P10D25:INT;
	P10D26:INT;
	P10D27:INT;
	P10D28:INT;
	P10D29:INT;
	P10D30:INT;
	P10STG:STRING;

END_VAR
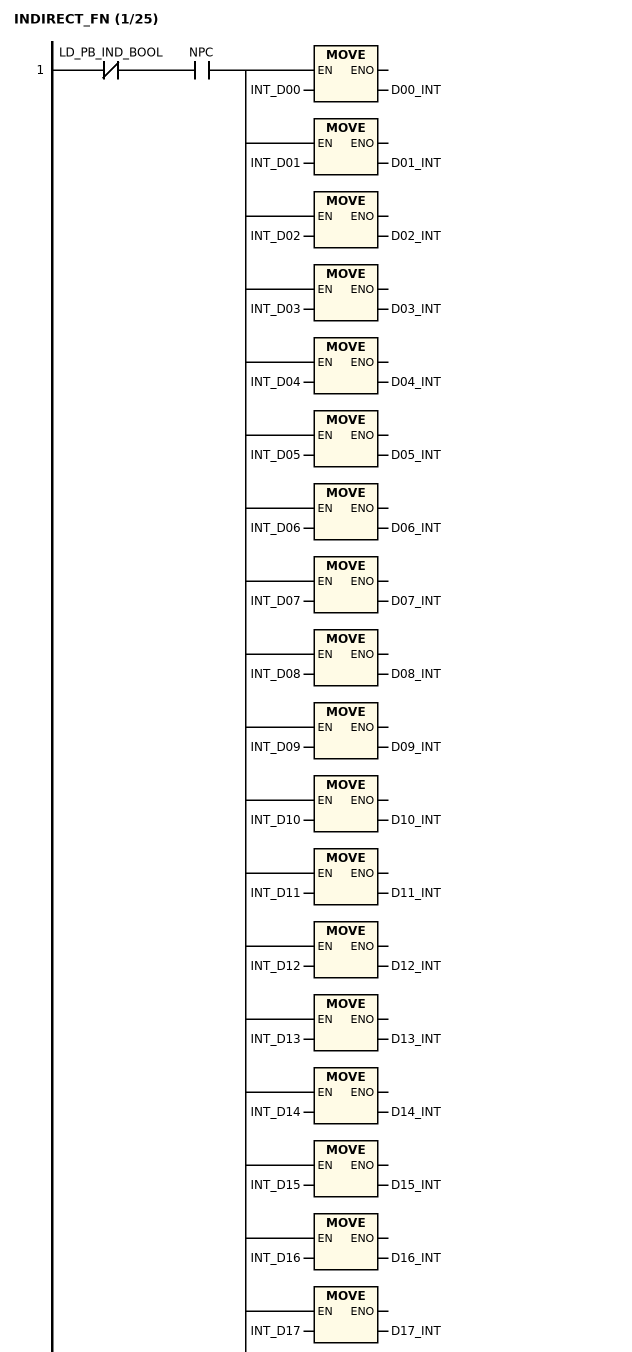
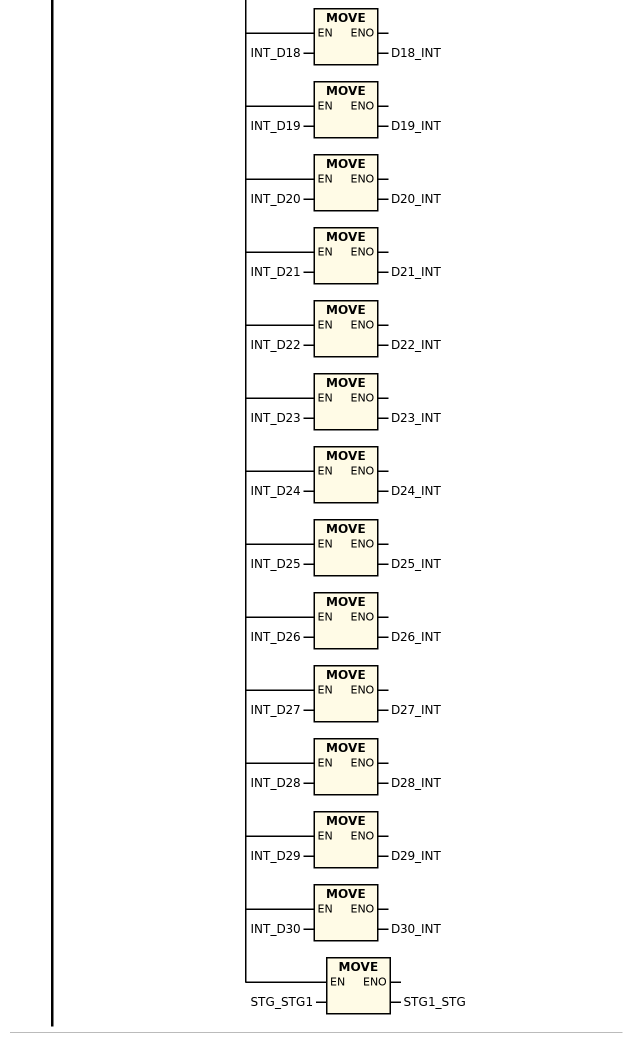
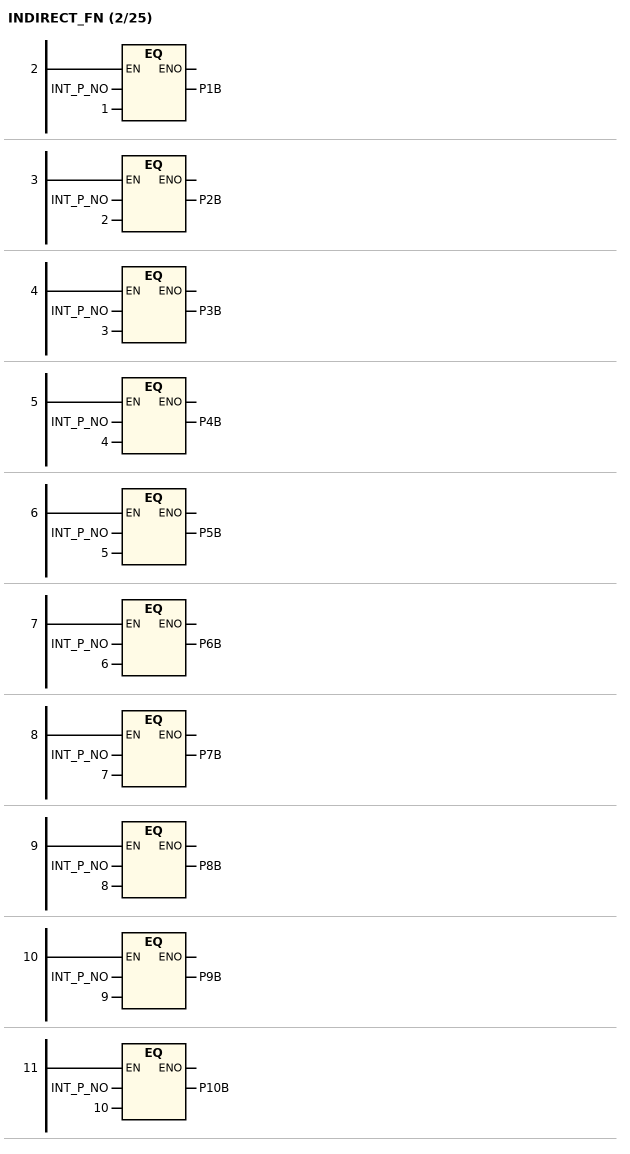
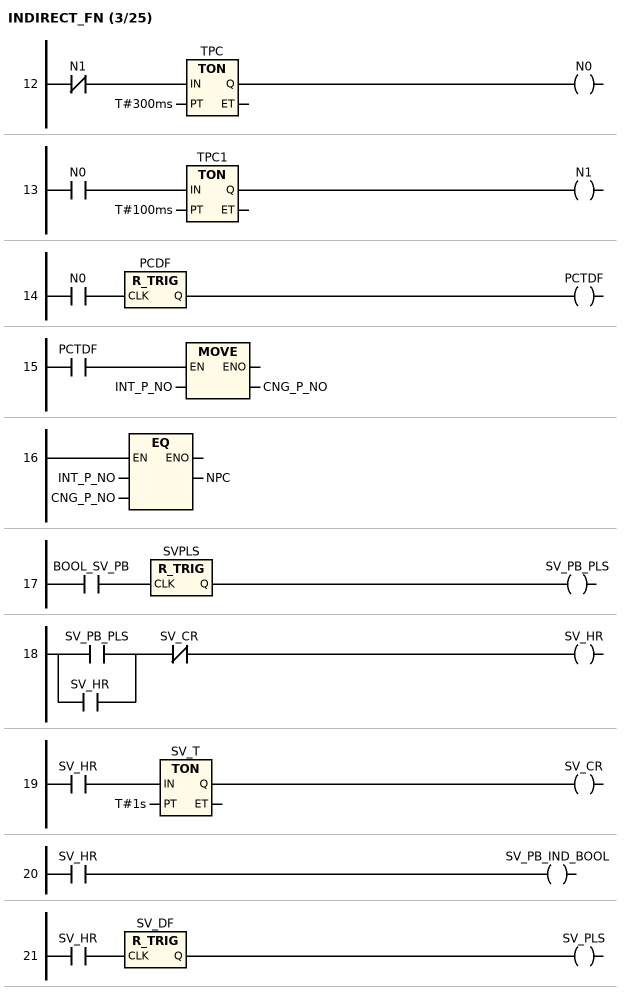
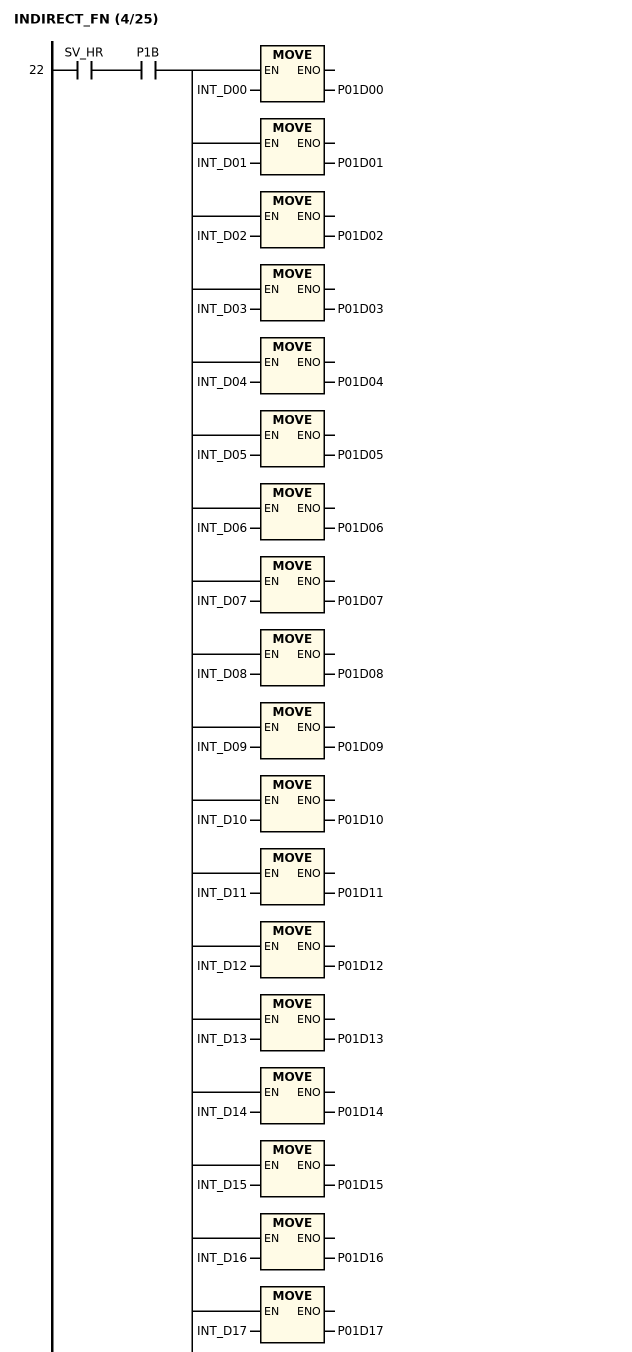
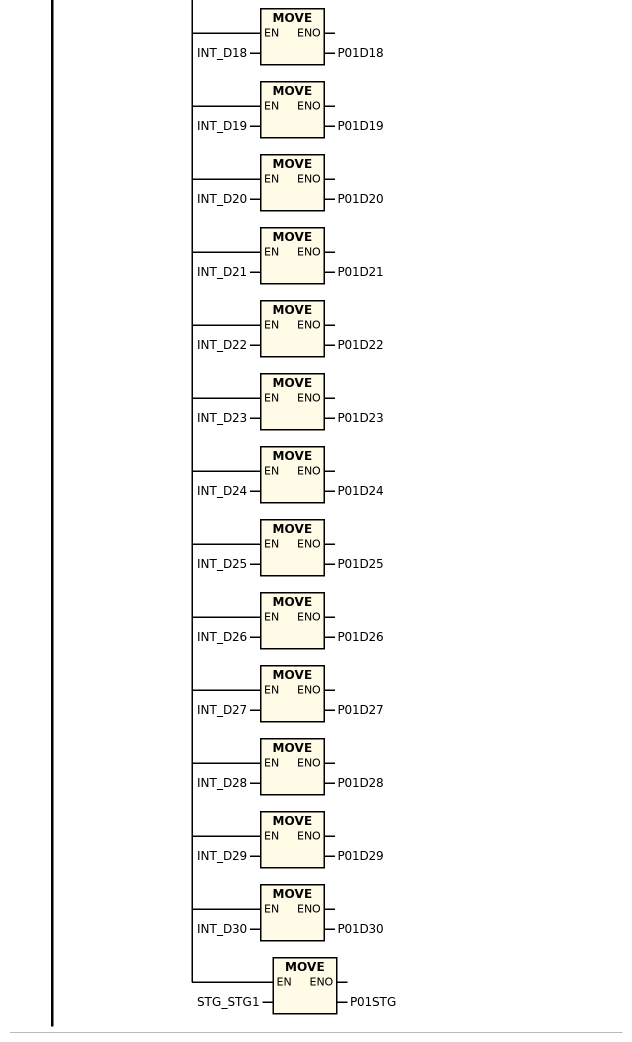
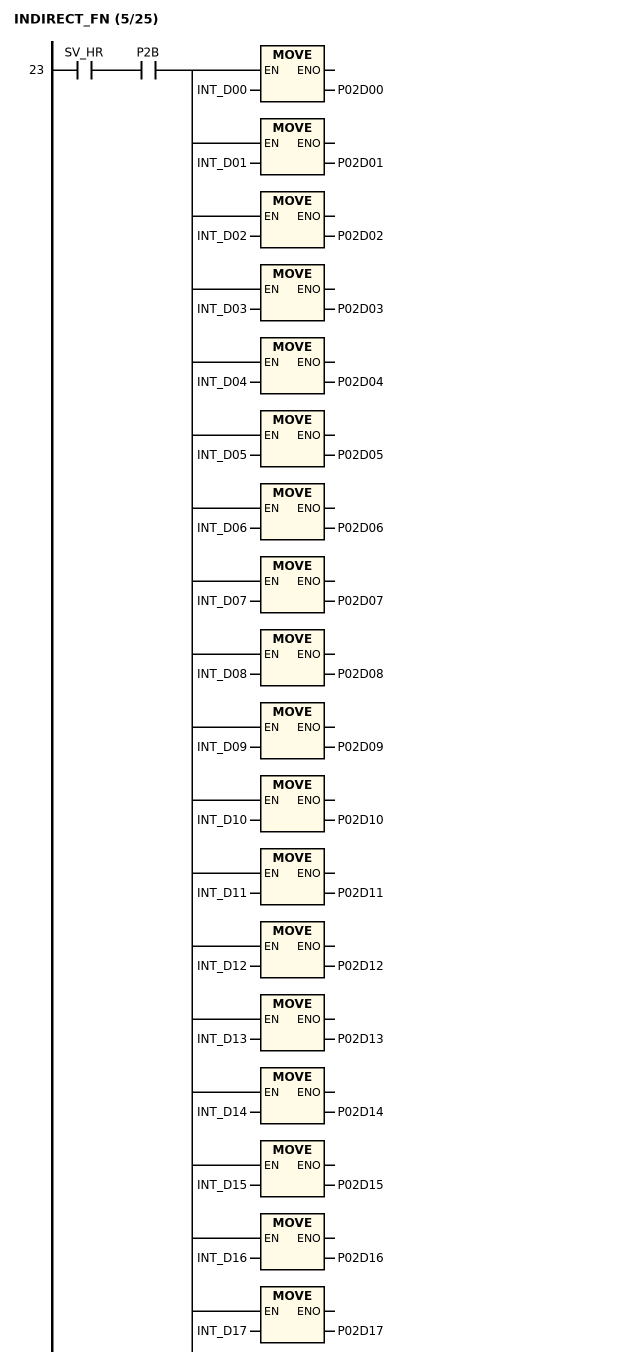
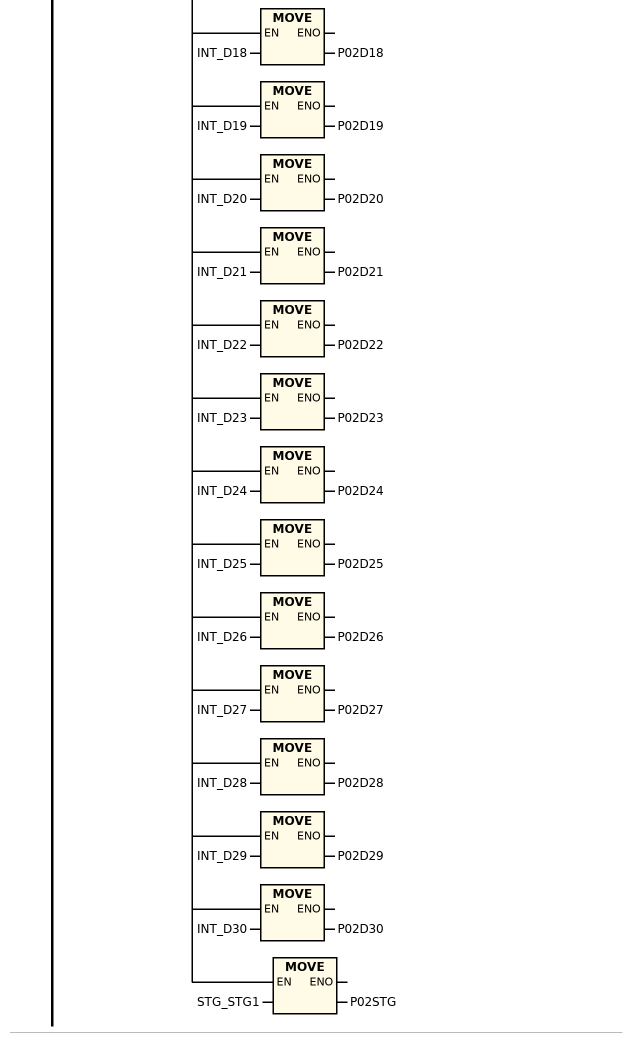
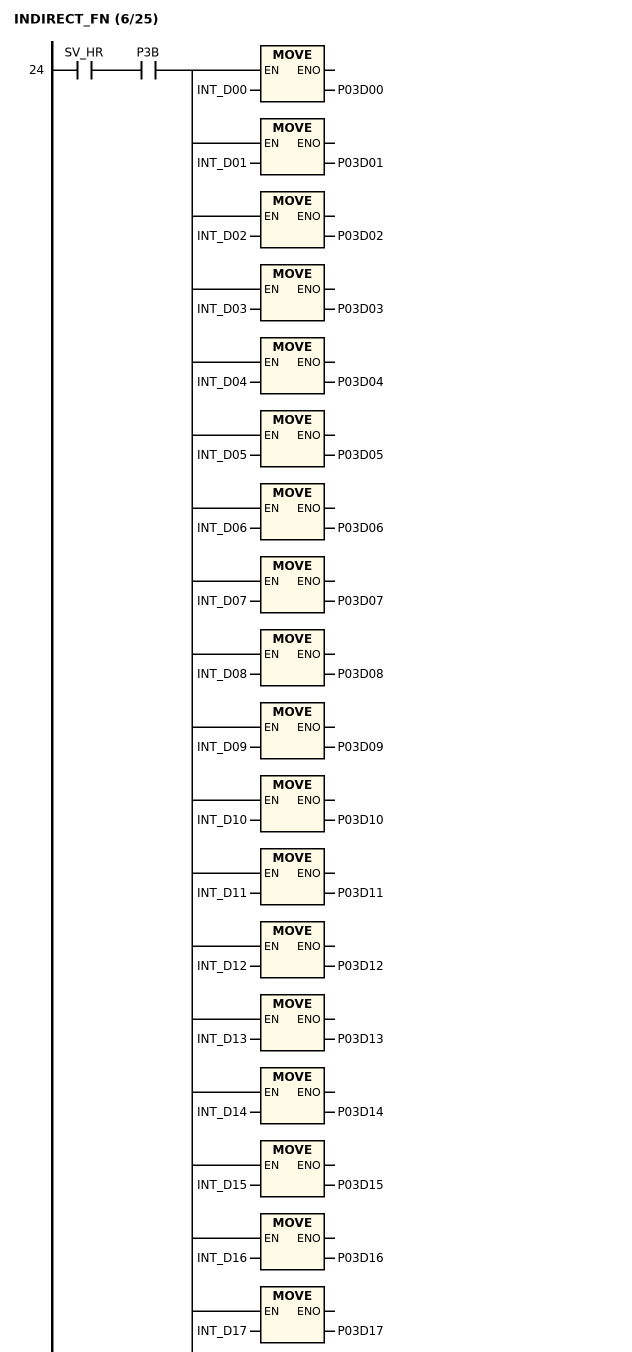
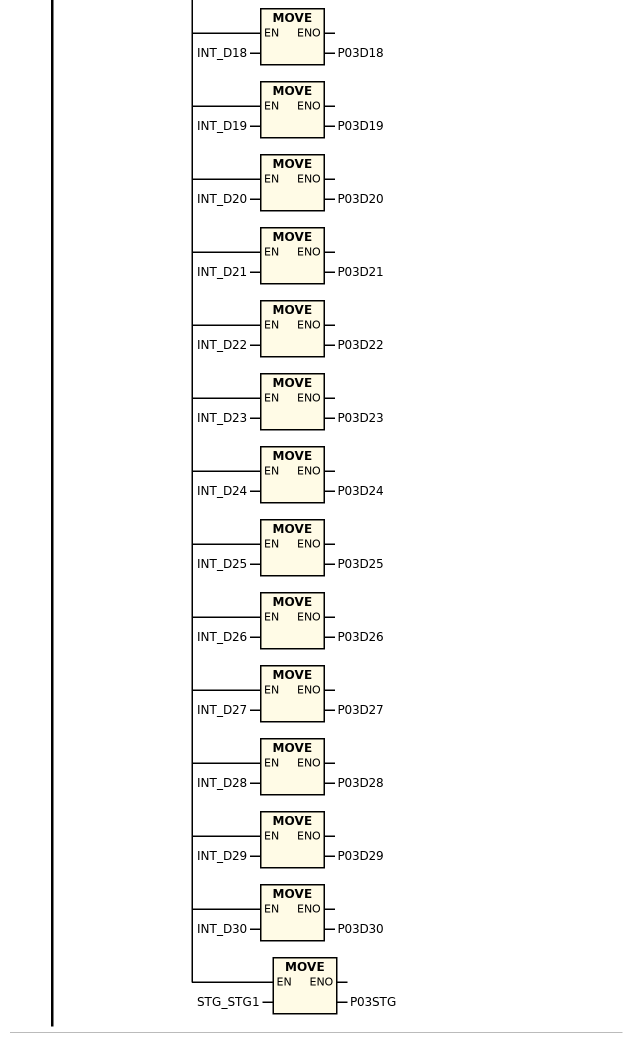
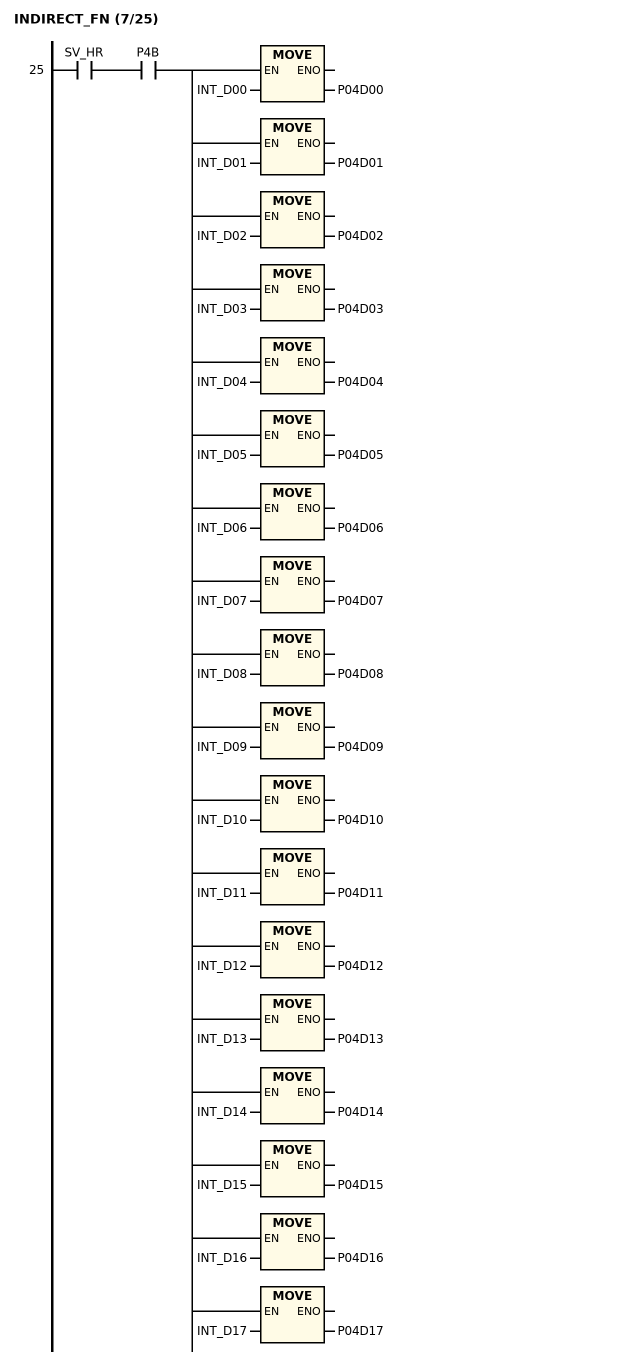
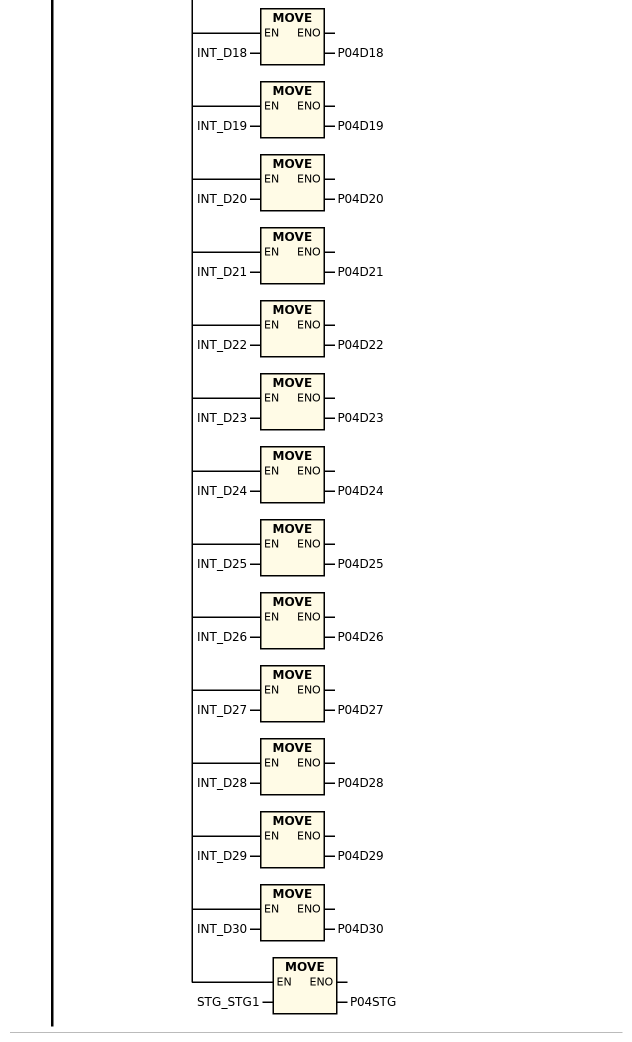
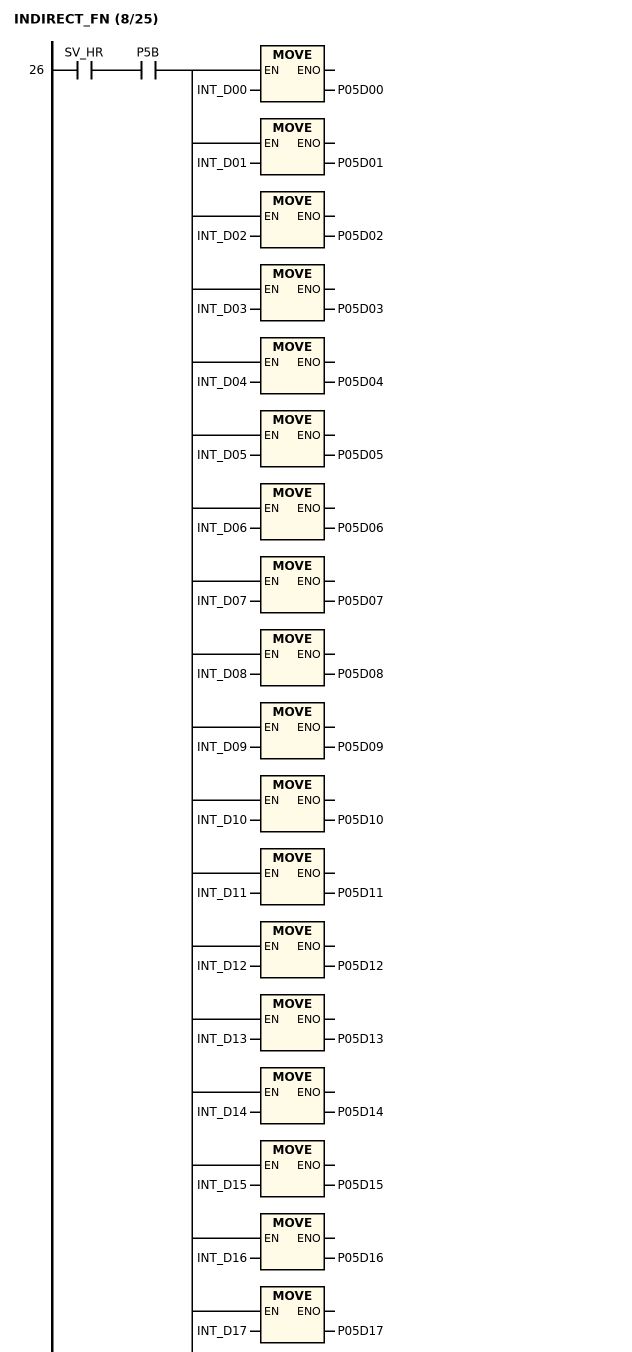
